// TwinCAT 3 PLC project Shutdown
// ProgramVersion: 3.1.4022.0
// libraries:
//   Tc2_Standard, * (Beckhoff Automation GmbH)
//   Tc2_System, * (Beckhoff Automation GmbH)
//   Tc2_Utilities, * (Beckhoff Automation GmbH)
//   Tc3_Module, * (Beckhoff Automation GmbH)
// project tree:
//   / PlcTask.TcTTO
//   POUs/ MAIN.TcPOU, Shutdown.TcPOU
// real-time tasks:
//   TASK PlcTask: cycle T#10ms, priority 20, ADS port 350
//   TASK updateIrSensors: cycle T#5ms, priority 9, ADS port 351
//   TASK UDP Task: cycle T#10ms, priority 10, ADS port 354
// motion (NC):
//   TASK NC-Task 1 SAF: cycle T#2ms, priority 4, ADS port 501
//   TASK NC-Task 1 SVB: cycle T#10ms, priority 8, ADS port 511
//   AXIS Achse 1 (id 1)
//     Velo: Maximum=20000
//     OtherSettings: AllowMotionCmdToSlave=true
//     encoder EncType=4
//       EncPara: ScaleFactorNumerator=0.01125, MaxCount=#x0000ffff
//         Inc: RefMode=2, RefSoftSyncMask=#x0000ffff
//         TimeComp: TimeCompMode=1, EncDelayCycles=4
//     drive DrvType=23
//       Analog: VeloReferenz=21600, ScaleFactorActTorque=0.1
//       TimeComp: TaskDelayCycles=1
//     controller CtrType=1
//       CtrPara: PriorControlFactor=1
//         PosDiffControl: Enable=false
//         Observer: BandWidth=20
//   AXIS Achse 2 (id 2)
//     Velo: Maximum=20000
//     OtherSettings: AllowMotionCmdToSlave=true
//     encoder EncType=4
//       EncPara: ScaleFactorNumerator=0.01125, MaxCount=#x0000ffff
//         Inc: RefSoftSyncMask=#x0000ffff
//         TimeComp: TimeCompMode=1, EncDelayCycles=4
//     drive DrvType=23
//       Analog: VeloReferenz=21600, ScaleFactorActTorque=0.1
//       TimeComp: TaskDelayCycles=1
//     controller CtrType=1
//       CtrPara: PriorControlFactor=1
//         PosDiffControl: Enable=false
//         Observer: BandWidth=20
//   AXIS Achse 3 (id 3)
//     Velo: Maximum=20000
//     OtherSettings: AllowMotionCmdToSlave=true
//     encoder EncType=4
//       EncPara: ScaleFactorNumerator=0.01125, MaxCount=#x0000ffff
//         Inc: RefSoftSyncMask=#x0000ffff
//         TimeComp: TimeCompMode=1, EncDelayCycles=4
//     drive DrvType=23
//       Analog: VeloReferenz=21600, ScaleFactorActTorque=0.1
//       TimeComp: TaskDelayCycles=1
//     controller CtrType=1
//       CtrPara: PriorControlFactor=1
//         PosDiffControl: Enable=false
//         Observer: BandWidth=20
//   AXIS Achse 4 (id 4)
//     OtherSettings: AllowMotionCmdToSlave=true
//     encoder EncType=4
//       EncPara: MaxCount=#x0000ffff
//         Inc: RefSoftSyncMask=#x0000ffff
//     drive DrvType=23
//       Analog: ScaleFactorActTorque=0.1
//       TimeComp: TaskDelayCycles=1
//     controller CtrType=1
//       CtrPara: PriorControlFactor=1
//         Observer: BandWidth=20
// I/O:
//   DEVICE Gerät 1 (EtherCAT), AmsNetId 5.49.201.214.2.1
//     Klemme 1 (EK1200) [EK1200-5000 EtherCAT Netzteil (2A E-Bus)]
//       Motorcontroller 1 [EL7342 2K. DC-Motor-Endstufe (50V, 3.5A)]
//       Motorcontroller 2 [EL7342 2K. DC-Motor-Endstufe (50V, 3.5A)]
//       8 Kanal Digital Input [EL1008 8K. Dig. Eingang 24V, 3ms]
//       4 Kanal Digital Output [EL2004 4K. Dig. Ausgang 24V, 0.5A]
//       8 Kanal Analog Input [EL3068 8K. Ana. Eingang 0-10V]
//       4 Kanal Analog Input [EL3064 4K.Ana. Eingang 0-10V]
//       Netzteilklemme 5V [EL9505 Netzteilklemme 5V]
//       Klemme 9 (EL9011) [EL9011 Endklemme]
//   DEVICE WLAN Adapter
// variable links:
//   Device 1 (EtherCAT) <-> irSensors/irSensors_Obj1 (updateIrSensors)
//     Term 1 (EK1200)/4 Kanal Analog Input/AI Standard Channel 1/IR Sensor 9 <-> Inputs/irInputData[8]
//     Term 1 (EK1200)/8 Kanal Analog Input/AI Standard Channel 1/IR Sensor 1 <-> Inputs/irInputData[0]
//     Term 1 (EK1200)/8 Kanal Analog Input/AI Standard Channel 2/IR Sensor 2 <-> Inputs/irInputData[1]
//     Term 1 (EK1200)/8 Kanal Analog Input/AI Standard Channel 3/IR Sensor 3 <-> Inputs/irInputData[2]
//     Term 1 (EK1200)/8 Kanal Analog Input/AI Standard Channel 4/IR Sensor 4 <-> Inputs/irInputData[3]
//     Term 1 (EK1200)/8 Kanal Analog Input/AI Standard Channel 5/IR Sensor 5 <-> Inputs/irInputData[4]
//     Term 1 (EK1200)/8 Kanal Analog Input/AI Standard Channel 6/IR Sensor 6 <-> Inputs/irInputData[5]
//     Term 1 (EK1200)/8 Kanal Analog Input/AI Standard Channel 7/IR Sensor 7 <-> Inputs/irInputData[6]
//     Term 1 (EK1200)/8 Kanal Analog Input/AI Standard Channel 8/IR Sensor 8 <-> Inputs/irInputData[7]
//   NC-Task 1 SAF/Axes/Achse 1 <-> Device 1 (EtherCAT)/Term 1 (EK1200)/Motorcontroller 1
//     Drive/Inputs/In/nState1 @bit 3 <-> DCM Status Channel 1/Status/Error
//     Drive/Inputs/In/nState1 @bit 5 <-> DCM Status Channel 1/Status/Moving negative
//     Drive/Inputs/In/nState1 @bit 4 <-> DCM Status Channel 1/Status/Moving positive
//     Drive/Inputs/In/nState1 @bit 1 <-> DCM Status Channel 1/Status/Ready
//     Drive/Inputs/In/nState1 <-> DCM Status Channel 1/Status/Ready to enable
//     Drive/Inputs/In/nState1 @bit 6 <-> DCM Status Channel 1/Status/Torque reduced
//     Drive/Inputs/In/nState1 @bit 2 <-> DCM Status Channel 1/Status/Warning
//     Drive/Inputs/In/nState2 @bit 3 <-> DCM Status Channel 1/Status/Digital input 1
//     Drive/Inputs/In/nState2 @bit 4 <-> DCM Status Channel 1/Status/Digital input 2
//     Drive/Inputs/In/nState2 @bit 5 <-> DCM Status Channel 1/Status/Sync error
//     Drive/Inputs/In/nState2 @bit 7 <-> DCM Status Channel 1/Status/TxPDO Toggle
//     Drive/Inputs/In/nState4 @bit 1 <-> WcState/InputToggle
//     Drive/Inputs/In/nState4 <-> WcState/WcState
//     Drive/Outputs/Out/nCtrl1 <-> DCM Control Channel 1/Control/Enable
//     Drive/Outputs/Out/nCtrl1 @bit 2 <-> DCM Control Channel 1/Control/Reduce torque
//     Drive/Outputs/Out/nCtrl1 @bit 1 <-> DCM Control Channel 1/Control/Reset
//     Drive/Outputs/Out/nDataOut2[0] <-> DCM Velocity Channel 1/Velocity
//     Enc/Inputs/In/nDataIn1[0] <-> ENC Status compact Channel 1/Counter value
//     Enc/Inputs/In/nDataIn2[0] <-> ENC Status compact Channel 1/Latch value
//     Enc/Inputs/In/nState1 @bit 4 <-> ENC Status compact Channel 1/Status/Counter overflow
//     Enc/Inputs/In/nState1 @bit 3 <-> ENC Status compact Channel 1/Status/Counter underflow
//     Enc/Inputs/In/nState1 @bit 7 <-> ENC Status compact Channel 1/Status/Extrapolation stall
//     Enc/Inputs/In/nState1 @bit 1 <-> ENC Status compact Channel 1/Status/Latch extern valid
//     Enc/Inputs/In/nState1 @bit 2 <-> ENC Status compact Channel 1/Status/Set counter done
//     Enc/Inputs/In/nState2 @bit 4 <-> ENC Status compact Channel 1/Status/Status of extern latch
//     Enc/Inputs/In/nState2 <-> ENC Status compact Channel 1/Status/Status of input A
//     Enc/Inputs/In/nState2 @bit 1 <-> ENC Status compact Channel 1/Status/Status of input B
//     Enc/Inputs/In/nState2 @bit 5 <-> ENC Status compact Channel 1/Status/Sync error
//     Enc/Inputs/In/nState2 @bit 7 <-> ENC Status compact Channel 1/Status/TxPDO Toggle
//     Enc/Inputs/In/nState4 @bit 1 <-> WcState/InputToggle
//     Enc/Inputs/In/nState4 <-> WcState/WcState
//     Enc/Outputs/Out/nCtrl1 @bit 3 <-> ENC Control compact Channel 1/Control/Enable latch extern on negative edge
//     Enc/Outputs/Out/nCtrl1 @bit 1 <-> ENC Control compact Channel 1/Control/Enable latch extern on positive edge
//     Enc/Outputs/Out/nCtrl1 @bit 2 <-> ENC Control compact Channel 1/Control/Set counter
//     Enc/Outputs/Out/nDataOut1[0] <-> ENC Control compact Channel 1/Set counter value
//   NC-Task 1 SAF/Axes/Achse 2 <-> Device 1 (EtherCAT)/Term 1 (EK1200)/Motorcontroller 1
//     Drive/Inputs/In/nState1 @bit 3 <-> DCM Status Channel 2/Status/Error
//     Drive/Inputs/In/nState1 @bit 5 <-> DCM Status Channel 2/Status/Moving negative
//     Drive/Inputs/In/nState1 @bit 4 <-> DCM Status Channel 2/Status/Moving positive
//     Drive/Inputs/In/nState1 @bit 1 <-> DCM Status Channel 2/Status/Ready
//     Drive/Inputs/In/nState1 <-> DCM Status Channel 2/Status/Ready to enable
//     Drive/Inputs/In/nState1 @bit 6 <-> DCM Status Channel 2/Status/Torque reduced
//     Drive/Inputs/In/nState1 @bit 2 <-> DCM Status Channel 2/Status/Warning
//     Drive/Inputs/In/nState2 @bit 3 <-> DCM Status Channel 2/Status/Digital input 1
//     Drive/Inputs/In/nState2 @bit 4 <-> DCM Status Channel 2/Status/Digital input 2
//     Drive/Inputs/In/nState2 @bit 5 <-> DCM Status Channel 2/Status/Sync error
//     Drive/Inputs/In/nState2 @bit 7 <-> DCM Status Channel 2/Status/TxPDO Toggle
//     Drive/Inputs/In/nState4 @bit 1 <-> WcState/InputToggle
//     Drive/Inputs/In/nState4 <-> WcState/WcState
//     Drive/Outputs/Out/nCtrl1 <-> DCM Control Channel 2/Control/Enable
//     Drive/Outputs/Out/nCtrl1 @bit 2 <-> DCM Control Channel 2/Control/Reduce torque
//     Drive/Outputs/Out/nCtrl1 @bit 1 <-> DCM Control Channel 2/Control/Reset
//     Drive/Outputs/Out/nDataOut2[0] <-> DCM Velocity Channel 2/Velocity
//     Enc/Inputs/In/nDataIn1[0] <-> ENC Status compact Channel 2/Counter value
//     Enc/Inputs/In/nDataIn2[0] <-> ENC Status compact Channel 2/Latch value
//     Enc/Inputs/In/nState1 @bit 4 <-> ENC Status compact Channel 2/Status/Counter overflow
//     Enc/Inputs/In/nState1 @bit 3 <-> ENC Status compact Channel 2/Status/Counter underflow
//     Enc/Inputs/In/nState1 @bit 7 <-> ENC Status compact Channel 2/Status/Extrapolation stall
//     Enc/Inputs/In/nState1 @bit 1 <-> ENC Status compact Channel 2/Status/Latch extern valid
//     Enc/Inputs/In/nState1 @bit 2 <-> ENC Status compact Channel 2/Status/Set counter done
//     Enc/Inputs/In/nState2 @bit 4 <-> ENC Status compact Channel 2/Status/Status of extern latch
//     Enc/Inputs/In/nState2 <-> ENC Status compact Channel 2/Status/Status of input A
//     Enc/Inputs/In/nState2 @bit 1 <-> ENC Status compact Channel 2/Status/Status of input B
//     Enc/Inputs/In/nState2 @bit 5 <-> ENC Status compact Channel 2/Status/Sync error
//     Enc/Inputs/In/nState2 @bit 7 <-> ENC Status compact Channel 2/Status/TxPDO Toggle
//     Enc/Inputs/In/nState4 @bit 1 <-> WcState/InputToggle
//     Enc/Inputs/In/nState4 <-> WcState/WcState
//     Enc/Outputs/Out/nCtrl1 @bit 3 <-> ENC Control compact Channel 2/Control/Enable latch extern on negative edge
//     Enc/Outputs/Out/nCtrl1 @bit 1 <-> ENC Control compact Channel 2/Control/Enable latch extern on positive edge
//     Enc/Outputs/Out/nCtrl1 @bit 2 <-> ENC Control compact Channel 2/Control/Set counter
//     Enc/Outputs/Out/nDataOut1[0] <-> ENC Control compact Channel 2/Set counter value
//   NC-Task 1 SAF/Axes/Achse 3 <-> Device 1 (EtherCAT)/Term 1 (EK1200)/Motorcontroller 2
//     Drive/Inputs/In/nState1 @bit 3 <-> DCM Status Channel 1/Status/Error
//     Drive/Inputs/In/nState1 @bit 5 <-> DCM Status Channel 1/Status/Moving negative
//     Drive/Inputs/In/nState1 @bit 4 <-> DCM Status Channel 1/Status/Moving positive
//     Drive/Inputs/In/nState1 @bit 1 <-> DCM Status Channel 1/Status/Ready
//     Drive/Inputs/In/nState1 <-> DCM Status Channel 1/Status/Ready to enable
//     Drive/Inputs/In/nState1 @bit 6 <-> DCM Status Channel 1/Status/Torque reduced
//     Drive/Inputs/In/nState1 @bit 2 <-> DCM Status Channel 1/Status/Warning
//     Drive/Inputs/In/nState2 @bit 3 <-> DCM Status Channel 1/Status/Digital input 1
//     Drive/Inputs/In/nState2 @bit 4 <-> DCM Status Channel 1/Status/Digital input 2
//     Drive/Inputs/In/nState2 @bit 5 <-> DCM Status Channel 1/Status/Sync error
//     Drive/Inputs/In/nState2 @bit 7 <-> DCM Status Channel 1/Status/TxPDO Toggle
//     Drive/Inputs/In/nState4 @bit 1 <-> WcState/InputToggle
//     Drive/Inputs/In/nState4 <-> WcState/WcState
//     Drive/Outputs/Out/nCtrl1 <-> DCM Control Channel 1/Control/Enable
//     Drive/Outputs/Out/nCtrl1 @bit 2 <-> DCM Control Channel 1/Control/Reduce torque
//     Drive/Outputs/Out/nCtrl1 @bit 1 <-> DCM Control Channel 1/Control/Reset
//     Drive/Outputs/Out/nDataOut2[0] <-> DCM Velocity Channel 1/Velocity
//     Enc/Inputs/In/nDataIn1[0] <-> ENC Status compact Channel 1/Counter value
//     Enc/Inputs/In/nDataIn2[0] <-> ENC Status compact Channel 1/Latch value
//     Enc/Inputs/In/nState1 @bit 4 <-> ENC Status compact Channel 1/Status/Counter overflow
//     Enc/Inputs/In/nState1 @bit 3 <-> ENC Status compact Channel 1/Status/Counter underflow
//     Enc/Inputs/In/nState1 @bit 7 <-> ENC Status compact Channel 1/Status/Extrapolation stall
//     Enc/Inputs/In/nState1 @bit 1 <-> ENC Status compact Channel 1/Status/Latch extern valid
//     Enc/Inputs/In/nState1 @bit 2 <-> ENC Status compact Channel 1/Status/Set counter done
//     Enc/Inputs/In/nState2 @bit 4 <-> ENC Status compact Channel 1/Status/Status of extern latch
//     Enc/Inputs/In/nState2 <-> ENC Status compact Channel 1/Status/Status of input A
//     Enc/Inputs/In/nState2 @bit 1 <-> ENC Status compact Channel 1/Status/Status of input B
//     Enc/Inputs/In/nState2 @bit 5 <-> ENC Status compact Channel 1/Status/Sync error
//     Enc/Inputs/In/nState2 @bit 7 <-> ENC Status compact Channel 1/Status/TxPDO Toggle
//     Enc/Inputs/In/nState4 @bit 1 <-> WcState/InputToggle
//     Enc/Inputs/In/nState4 <-> WcState/WcState
//     Enc/Outputs/Out/nCtrl1 @bit 3 <-> ENC Control compact Channel 1/Control/Enable latch extern on negative edge
//     Enc/Outputs/Out/nCtrl1 @bit 1 <-> ENC Control compact Channel 1/Control/Enable latch extern on positive edge
//     Enc/Outputs/Out/nCtrl1 @bit 2 <-> ENC Control compact Channel 1/Control/Set counter
//     Enc/Outputs/Out/nDataOut1[0] <-> ENC Control compact Channel 1/Set counter value
//   NC-Task 1 SAF/Axes/Achse 4 <-> Device 1 (EtherCAT)/Term 1 (EK1200)/Motorcontroller 2
//     Drive/Inputs/In/nState1 @bit 3 <-> DCM Status Channel 2/Status/Error
//     Drive/Inputs/In/nState1 @bit 5 <-> DCM Status Channel 2/Status/Moving negative
//     Drive/Inputs/In/nState1 @bit 4 <-> DCM Status Channel 2/Status/Moving positive
//     Drive/Inputs/In/nState1 @bit 1 <-> DCM Status Channel 2/Status/Ready
//     Drive/Inputs/In/nState1 <-> DCM Status Channel 2/Status/Ready to enable
//     Drive/Inputs/In/nState1 @bit 6 <-> DCM Status Channel 2/Status/Torque reduced
//     Drive/Inputs/In/nState1 @bit 2 <-> DCM Status Channel 2/Status/Warning
//     Drive/Inputs/In/nState2 @bit 3 <-> DCM Status Channel 2/Status/Digital input 1
//     Drive/Inputs/In/nState2 @bit 4 <-> DCM Status Channel 2/Status/Digital input 2
//     Drive/Inputs/In/nState2 @bit 5 <-> DCM Status Channel 2/Status/Sync error
//     Drive/Inputs/In/nState2 @bit 7 <-> DCM Status Channel 2/Status/TxPDO Toggle
//     Drive/Inputs/In/nState4 @bit 1 <-> WcState/InputToggle
//     Drive/Inputs/In/nState4 <-> WcState/WcState
//     Drive/Outputs/Out/nCtrl1 <-> DCM Control Channel 2/Control/Enable
//     Drive/Outputs/Out/nCtrl1 @bit 2 <-> DCM Control Channel 2/Control/Reduce torque
//     Drive/Outputs/Out/nCtrl1 @bit 1 <-> DCM Control Channel 2/Control/Reset
//     Drive/Outputs/Out/nDataOut2[0] <-> DCM Velocity Channel 2/Velocity
//     Enc/Inputs/In/nDataIn1[0] <-> ENC Status compact Channel 2/Counter value
//     Enc/Inputs/In/nDataIn2[0] <-> ENC Status compact Channel 2/Latch value
//     Enc/Inputs/In/nState1 @bit 4 <-> ENC Status compact Channel 2/Status/Counter overflow
//     Enc/Inputs/In/nState1 @bit 3 <-> ENC Status compact Channel 2/Status/Counter underflow
//     Enc/Inputs/In/nState1 @bit 7 <-> ENC Status compact Channel 2/Status/Extrapolation stall
//     Enc/Inputs/In/nState1 @bit 1 <-> ENC Status compact Channel 2/Status/Latch extern valid
//     Enc/Inputs/In/nState1 @bit 2 <-> ENC Status compact Channel 2/Status/Set counter done
//     Enc/Inputs/In/nState2 @bit 4 <-> ENC Status compact Channel 2/Status/Status of extern latch
//     Enc/Inputs/In/nState2 <-> ENC Status compact Channel 2/Status/Status of input A
//     Enc/Inputs/In/nState2 @bit 1 <-> ENC Status compact Channel 2/Status/Status of input B
//     Enc/Inputs/In/nState2 @bit 5 <-> ENC Status compact Channel 2/Status/Sync error
//     Enc/Inputs/In/nState2 @bit 7 <-> ENC Status compact Channel 2/Status/TxPDO Toggle
//     Enc/Inputs/In/nState4 @bit 1 <-> WcState/InputToggle
//     Enc/Inputs/In/nState4 <-> WcState/WcState
//     Enc/Outputs/Out/nCtrl1 @bit 3 <-> ENC Control compact Channel 2/Control/Enable latch extern on negative edge
//     Enc/Outputs/Out/nCtrl1 @bit 1 <-> ENC Control compact Channel 2/Control/Enable latch extern on positive edge
//     Enc/Outputs/Out/nCtrl1 @bit 2 <-> ENC Control compact Channel 2/Control/Set counter
//     Enc/Outputs/Out/nDataOut1[0] <-> ENC Control compact Channel 2/Set counter value
//   Shutdown/Shutdown Instance <-> Device 1 (EtherCAT)/Term 1 (EK1200)/8 Kanal Digital Input
//     PlcTask Inputs/Shutdown.bStart <-> Channel 8/Shutdown

CONFIGURATION Shutdown
    RESOURCE PLC ON TwinCAT3
        TASK PlcTask(INTERVAL := T#50000us, PRIORITY := 2);
        PROGRAM MAIN WITH PlcTask : MAIN;
    END_RESOURCE
END_CONFIGURATION

// ---- POUs/MAIN.TcPOU
PROGRAM MAIN
VAR
END_VAR

Shutdown();

END_PROGRAM

// ---- POUs/Shutdown.TcPOU
PROGRAM Shutdown
VAR
	bStart	AT%I* : BOOL := FALSE;
	Shutdown_Block: NT_Shutdown;
END_VAR

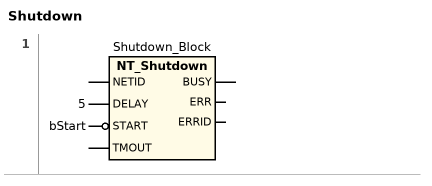
// NETWORK 1
Shutdown_Block(DELAY := 5, START := NOT bStart); // NT_Shutdown

END_PROGRAM
